SUBAPPLICATION A2X2_ILOCK_SWITCH_PROTECT (* Buendelt den NET-Roundtrip (bidirektionales A2X2) mit der Last-Wins-Arbitrierung samt Schutz-Totzeit: A2X2_TO_A2X spaltet A2X2 in ein unidirektionales A2X-Socket (Taster-Zustand) + -Plug (Rueckschreibe-Zustand), ILOCK_SWITCH_PROTECT_A2X arbeitet direkt auf dem gebuendelten Paar, A2X_SPLIT_2 dupliziert den interlocked Zustand auf den Rueckschreibe-Pfad und auf den externen A2X-Plug (fuer die physischen Ausgaenge) - 'SUB style': Bridge+Interlock+Split stecken im Composite, nicht in der Resource des Geraets. *)
  (* Standard: 61499-2; Description: Copyright (c) 2026 HR Agrartechnik GmbH This program and the accompanying materials are made available under the terms of the Eclipse Public License 2.0 which is available at https://www.eclipse.org/legal/epl-2.0/ SPDX-License-Identifier: EPL-2.0 *)
  (* Version 1.0, 2026-09-05, Franz Höpfinger, HR Agrartechnik GmbH, initial API and implementation and/or initial documentation *)
  PACKAGE MyLib::sys;
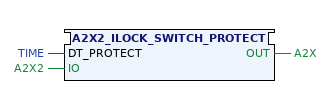
  VAR_INPUT
    DT_PROTECT : TIME := T#50ms; (* Schutz-Totzeit vor Richtungswechsel *)
  END_VAR
  SOCKETS
    IO : adapter::types::bidirectional::A2X2; (* Gebuendelter NET-Roundtrip: Taster-Zustand rein, Rueckschreibe-Zustand raus *)
  END_SOCKETS
  PLUGS
    OUT : adapter::types::unidirectional::A2X; (* Interlocked UP/DOWN Zustand, fuer physische Ausgaenge *)
  END_PLUGS
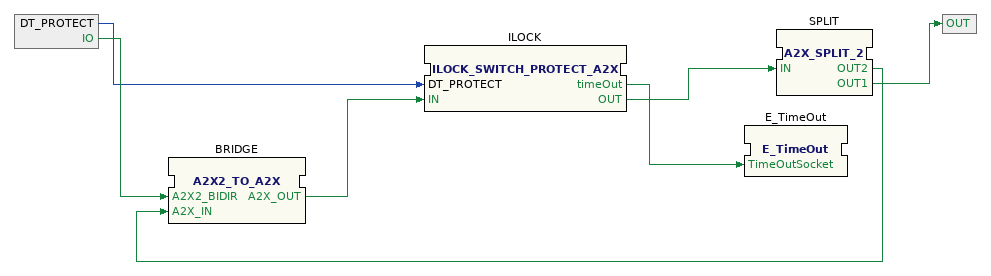
  FBS
    BRIDGE : adapter::conversion::bidirectional::A2X2_TO_A2X;
    ILOCK : logiBUS::signalprocessing::interlock::ILOCK_SWITCH_PROTECT_A2X;
    E_TimeOut : iec61499::events::E_TimeOut;
    SPLIT : adapter::events::unidirectional::A2X_SPLIT_2;
  END_FBS
  DATA_CONNECTIONS
    DT_PROTECT TO ILOCK.DT_PROTECT;
  END_CONNECTIONS
  ADAPTER_CONNECTIONS
    IO TO BRIDGE.A2X2_BIDIR;
    BRIDGE.A2X_OUT TO ILOCK.IN;
    ILOCK.timeOut TO E_TimeOut.TimeOutSocket;
    ILOCK.OUT TO SPLIT.IN;
    SPLIT.OUT2 TO BRIDGE.A2X_IN;
    SPLIT.OUT1 TO OUT;
  END_CONNECTIONS
END_SUBAPPLICATION
